(* CoDeSys 2.3.9.59 project: TwinCATRx.pro *)
(* Libraries: STANDARD.LIB *)

(* Task configuration *)
TASK Standard (PRIORITY := 0, INTERVAL := T#1ms);
	MAIN
END_TASK

(* Global variable list: Global_Variables *)
VAR_GLOBAL
(* Simple types *)
	AString			: STRING;
	ABool			: BOOL;
	AByte			: BYTE;
	AInt				: INT;
	ADInt			: DINT;
	(*ALInt			: LINT;*)
	AReal			: REAL;
	ALReal			: LREAL;
(* Arrays *)
	ArrString			: ARRAY [0..10] OF STRING;
	ArrBool			: ARRAY [0..10] OF BOOL;
	ArrByte			: ARRAY [0..10] OF BYTE;
	ArrInt			: ARRAY [0..10] OF INT;
	ArrDInt			: ARRAY [0..10] OF DINT;
	(*ArrLInt			: ARRAY [0..10] OF LINT;*)
	ArrReal			: ARRAY [0..10] OF REAL;
	ArrLReal			: ARRAY [0..10] OF LREAL;
(* Structures *)
	Tag1			: STRUCT_Object;
	Tag2			: STRUCT_Object2;
	Tag3			: STRUCT_Object3;
(* Hardware Mappings *)
	Out1				AT %QX0.0	: BOOL;
	Out2				AT %QX0.1	: BOOL;
	Out3				AT %QX0.2	: BOOL;
	Out4				AT %QX0.3	: BOOL;
END_VAR

(* Data type *)
TYPE STRUCT_Object :
STRUCT
(* Simple types *)
	AString			: STRING;
	ABool			: BOOL;
	AByte			: BYTE;
	AInt				: INT;
	ADInt			: DINT;
	(*ALInt			: LINT;*)
	AReal			: REAL;
	ALReal			: LREAL;
(* Structure in a structure *)
	Object2			: STRUCT_Object2;
END_STRUCT
END_TYPE

(* Data type *)
TYPE STRUCT_Object2 :
STRUCT
(* Simple types *)
	AString			: STRING;
	ABool			: BOOL;
	AByte			: BYTE;
	AInt				: INT;
	ADInt			: DINT;
	(*ALInt			: LINT;*)
	AReal			: REAL;
	ALReal			: LREAL;
	(*Object3			: STRUCT_Object3;*)
END_STRUCT
END_TYPE

(* Data type *)
TYPE STRUCT_Object3 :
STRUCT
(* Arrays *)
	ArrString			: ARRAY [0..10] OF STRING;
	ArrBool			: ARRAY [0..10] OF BOOL;
	ArrByte			: ARRAY [0..10] OF BYTE;
	ArrInt			: ARRAY [0..10] OF INT;
	ArrDInt			: ARRAY [0..10] OF DINT;
	(*ArrLInt			: ARRAY [0..10] OF LINT;*)
	ArrReal			: ARRAY [0..10] OF REAL;
	ArrLReal			: ARRAY [0..10] OF LREAL;
END_STRUCT
END_TYPE

(* POU MAIN, ST *)
PROGRAM MAIN
VAR
END_VAR
;
END_PROGRAM
